// TIA Portal V21 export
DATA_BLOCK "FB_Read_Bits_From_Word_DB"   // DB23
AUTHOR : JEBU
FAMILY : VTEMdc
VERSION : 1.1
// stored: InstanceOfName FB_Read_Bits_From_Word, InstanceOfType FB
"FB_Read_Bits_From_Word"
   // VAR_INPUT
   //    wData { ExternalVisible := 'False'} : Word := 16#7510;
   //    iStartBit { ExternalVisible := 'False'} : Int := 0;
   //    iEndBit { ExternalVisible := 'False'} : Int := 15;
   // END_VAR
   // VAR_OUTPUT
   //    iValue { ExternalVisible := 'False'} : Int := 4213;
   //    xError { ExternalVisible := 'False'} : Bool := FALSE;
   // END_VAR
BEGIN
END_DATA_BLOCK
